// TIA Portal V20 export
DATA_BLOCK "DB_Valve1"   // DB2
TITLE = DB_Valve1
AUTHOR : Gemini
// stored: InstanceOfName FB_ValveControl, InstanceOfType FB
"FB_ValveControl"
   // VAR_INPUT
   //    bOpen : Bool;
   //    bClose : Bool;
   // END_VAR
   // VAR_OUTPUT
   //    bOpened : Bool;
   //    bClosed : Bool;
   //    bFault : Bool;
   // END_VAR
BEGIN
END_DATA_BLOCK
